TYPE CM_Valve_WRN :
STRUCT
END_STRUCT
END_TYPE

(* stored: Version 1.1.0.1, ProductVersion 3.1.4024.12
   DUT CM_Valve_WRN: Id {22a0f40a-9e7d-4c45-9796-98259d72e739} *)
